// TwinCAT 3 PLC project Elevator
// ProgramVersion: 3.1.4023.0
// libraries:
//   Tc2_Standard, * (Beckhoff Automation GmbH)
//   Tc3_Module, * (Beckhoff Automation GmbH)
// project tree:
//   Global Vars/ GVL.TcGVL
//   / PlcTask.TcTTO (not stored)
//   PRG/ FB_Elevator.TcPOU (not stored), MAIN.TcPOU
//   TASKS/ PlcTask.TcTTO (not stored)
//   UDT/ E_States.TcDUT (not stored), ST_Floor.TcDUT (not stored)
// real-time tasks:
//   TASK PlcTask: cycle T#10ms, priority 20, ADS port 350

// ---- Global Vars/GVL.TcGVL
VAR_GLOBAL
	Elevator:FB_Elevator;
	Floors:ARRAY[1..4]	OF	ST_Floor;
	RequestedFloor: INT;
	ActualFloor: INT;
END_VAR

// ---- PRG/MAIN.TcPOU
PROGRAM MAIN
VAR
	//Elevator:FB_Elevator;
	//Floors:ARRAY[1..4]	OF	ST_Floor;
	State: E_States;
	i: INT;
	//RequestedFloor: INT;
	//ActualFloor: INT;
	Trigger:ARRAY[1..4]	OF	R_TRIG;
END_VAR

CASE	State	OF
	E_States.Call:
		FOR	i:=1	TO	4	DO
			IF	Floors[i].Call	THEN
				RequestedFloor:=i;
			END_IF
		END_FOR
		
		IF	RequestedFloor>ActualFloor	THEN
			State:=E_States.MoveUp;	
		ELSIF	RequestedFloor<ActualFloor	THEN
			State:=E_States.MoveDown;	
		END_IF
	E_States.MoveUp:
		Elevator.MoveUp();
		FOR	i:=1	TO	4	DO
			Trigger[i](clk:=Floors[i].Low);
			IF	Trigger[i].Q	THEN
				ActualFloor:=ActualFloor+1;
			END_IF
		END_FOR
		
		IF	ActualFloor=RequestedFloor	THEN
			State:=E_States.SlowDown;
		END_IF
	E_States.MoveDown:
		Elevator.MoveDown();
		FOR	i:=1	TO	4	DO
			Trigger[i](clk:=Floors[i].High);
			IF	Trigger[i].Q	THEN
				ActualFloor:=ActualFloor-1;
			END_IF
		END_FOR
		
		IF	ActualFloor=RequestedFloor	THEN
			State:=E_States.SlowDown;
		END_IF
		
	E_States.SlowDown:
		Elevator.SlowDown();
		FOR	i:=1	TO	4	DO
			IF	Floors[i].Mid	THEN
				State:=E_States.Stop;
			END_IF
		END_FOR
	E_States.Stop:
		Elevator.Stop();
		State:=E_States.Call;
END_CASE

END_PROGRAM
